Universal Robots PolyScope program: paganini.urp

Program paganini (installation=string_planes directory=/programs/hard_coded_pieces createdIn=5.17.3 lastSavedIn=5.17.3 robotSerialNumber=20245501435)
Calibrated DH parameters: a=[0.000154, -0.137004, -0.385524, -0.00002, 0.000092, 0]; d=[0.162441, 211.794786, -230.585024, 18.923638, 0.099786, 0.09951]; alpha=[1.569493, -0.001902, 0.003874, 1.570111, -1.570167, 0]; deltaTheta=[0, -1.242934, 1.056292, 0.186646, 0.000002, 0.000001]
InitVariablesNode
Robot Program (runOnlyOnce=true)
  SuppressedNode
    Wait Sleep waitTime=30
  Timer (action=Start) variable(name=beats)
  MoveL speed 600 mm/s, acceleration 1000 mm/s^2 (useActiveTCP=true) feature=Base
    Waypoint a_tip: TCP in base x=525.206 y=350.983 z=214.78 mm, rx=-1.3698 ry=-2.3362 rz=1.327 rad; joints [-161.028, -44.56, 81.191, -78.693, -115.03, -178.818] deg; TCP offset x=28.21 y=-96.107 z=-99.69 mm, rx=0 ry=0 rz=0 rad
    Waypoint a_frog: TCP in base x=336.638 y=773.336 z=103.937 mm, rx=-1.3698 ry=-2.3362 rz=1.327 rad; joints [-127.102, -6.181, 18.995, -50.118, -88.699, -156.884] deg
      Until EXPRESSION (allowActions=false) ExpressionBranch=beats≥1
    SuppressedNode
      Popup Message (haltProgram=false inputType=Variable) variable=beats
    Timer (action=Reset) variable=beats
  MoveL speed 150 mm/s, acceleration 400 mm/s^2 (useActiveTCP=true) feature=Base
    Waypoint a_tip: TCP in base x=525.206 y=350.983 z=214.78 mm, rx=-1.3698 ry=-2.3362 rz=1.327 rad; joints [-161.028, -44.56, 81.191, -78.693, -115.03, -178.818] deg
      Until EXPRESSION (allowActions=false) ExpressionBranch=beats≥2.5
    Timer (action=Reset) variable=beats
  MoveL speed 200 mm/s, acceleration 1200 mm/s^2 (useActiveTCP=true) feature=Base
    Waypoint a_tip: TCP in base x=525.206 y=350.983 z=214.78 mm, rx=-1.3698 ry=-2.3362 rz=1.327 rad; joints [-161.028, -44.56, 81.191, -78.693, -115.03, -178.818] deg
      Until EXPRESSION (allowActions=false) ExpressionBranch=beats≥0.75
    Timer (action=Reset) variable=beats
  MoveL speed 150 mm/s, acceleration 400 mm/s^2 (useActiveTCP=true) feature=Base
    Waypoint a_frog: TCP in base x=336.638 y=773.336 z=103.937 mm, rx=-1.3698 ry=-2.3362 rz=1.327 rad; joints [-127.102, -6.181, 18.995, -50.118, -88.699, -156.884] deg
      Until EXPRESSION (allowActions=false) ExpressionBranch=beats≥2.5
    Timer (action=Reset) variable=beats
  MoveL speed 250 mm/s, acceleration 1200 mm/s^2 (useActiveTCP=true) feature=Base
    Waypoint a_frog: TCP in base x=336.638 y=773.336 z=103.937 mm, rx=-1.3698 ry=-2.3362 rz=1.327 rad; joints [-127.102, -6.181, 18.995, -50.118, -88.699, -156.884] deg
      Until EXPRESSION (allowActions=false) ExpressionBranch=beats≥0.75
    Timer (action=Reset) variable=beats
  MoveL speed 250 mm/s, acceleration 1200 mm/s^2 (useActiveTCP=true) feature=Base
    Waypoint a_tip: TCP in base x=525.206 y=350.983 z=214.78 mm, rx=-1.3698 ry=-2.3362 rz=1.327 rad; joints [-161.028, -44.56, 81.191, -78.693, -115.03, -178.818] deg
      Until EXPRESSION (allowActions=false) ExpressionBranch=beats≥0.75
    Timer (action=Reset) variable=beats
  MoveJ speed 100 deg/s, acceleration 100 deg/s^2 (useActiveTCP=true) feature=Base
    Waypoint a_frog: TCP in base x=336.638 y=773.336 z=103.937 mm, rx=-1.3698 ry=-2.3362 rz=1.327 rad; joints [-127.102, -6.181, 18.995, -50.118, -88.699, -156.884] deg
  Timer (action=Reset) variable=beats
  MoveL speed 200 mm/s, acceleration 200 mm/s^2 (useActiveTCP=true) feature=Base
    Waypoint a_tip: TCP in base x=525.206 y=350.983 z=214.78 mm, rx=-1.3698 ry=-2.3362 rz=1.327 rad; joints [-161.028, -44.56, 81.191, -78.693, -115.03, -178.818] deg
      Until EXPRESSION (allowActions=false) ExpressionBranch=beats≥3
    Timer (action=Reset) variable=beats
  MoveL speed 600 mm/s, acceleration 1000 mm/s^2 (useActiveTCP=true) feature=Base
    Waypoint a_frog: TCP in base x=336.638 y=773.336 z=103.937 mm, rx=-1.3698 ry=-2.3362 rz=1.327 rad; joints [-127.102, -6.181, 18.995, -50.118, -88.699, -156.884] deg
      Until EXPRESSION (allowActions=false) ExpressionBranch=beats≥1
    Timer (action=Reset) variable=beats
  MoveL speed 150 mm/s, acceleration 400 mm/s^2 (useActiveTCP=true) feature=Base
    Waypoint a_tip: TCP in base x=525.206 y=350.983 z=214.78 mm, rx=-1.3698 ry=-2.3362 rz=1.327 rad; joints [-161.028, -44.56, 81.191, -78.693, -115.03, -178.818] deg
      Until EXPRESSION (allowActions=false) ExpressionBranch=beats≥2.5
    Timer (action=Reset) variable=beats
  MoveL speed 250 mm/s, acceleration 1200 mm/s^2 (useActiveTCP=true) feature=Base
    Waypoint a_tip: TCP in base x=525.206 y=350.983 z=214.78 mm, rx=-1.3698 ry=-2.3362 rz=1.327 rad; joints [-161.028, -44.56, 81.191, -78.693, -115.03, -178.818] deg
      Until EXPRESSION (allowActions=false) ExpressionBranch=beats≥0.75
    Timer (action=Reset) variable=beats
  MoveL speed 150 mm/s, acceleration 400 mm/s^2 (useActiveTCP=true) feature=Base
    Waypoint a_frog: TCP in base x=336.638 y=773.336 z=103.937 mm, rx=-1.3698 ry=-2.3362 rz=1.327 rad; joints [-127.102, -6.181, 18.995, -50.118, -88.699, -156.884] deg
      Until EXPRESSION (allowActions=false) ExpressionBranch=beats≥1.5
    Timer (action=Reset) variable=beats
  MoveL speed 250 mm/s, acceleration 1200 mm/s^2 (useActiveTCP=true) feature=Base
    Waypoint a_tip: TCP in base x=525.206 y=350.983 z=214.78 mm, rx=-1.3698 ry=-2.3362 rz=1.327 rad; joints [-161.028, -44.56, 81.191, -78.693, -115.03, -178.818] deg
      Until EXPRESSION (allowActions=false) ExpressionBranch=beats≥0.75
    Timer (action=Reset) variable=beats
  MoveL speed 150 mm/s, acceleration 400 mm/s^2 (useActiveTCP=true) feature=Base
    Waypoint a_frog: TCP in base x=336.638 y=773.336 z=103.937 mm, rx=-1.3698 ry=-2.3362 rz=1.327 rad; joints [-127.102, -6.181, 18.995, -50.118, -88.699, -156.884] deg
      Until EXPRESSION (allowActions=false) ExpressionBranch=beats≥1.5
    Timer (action=Reset) variable=beats
  MoveL speed 250 mm/s, acceleration 1200 mm/s^2 (useActiveTCP=true) feature=Base
    Waypoint a_frog: TCP in base x=336.638 y=773.336 z=103.937 mm, rx=-1.3698 ry=-2.3362 rz=1.327 rad; joints [-127.102, -6.181, 18.995, -50.118, -88.699, -156.884] deg
      Until EXPRESSION (allowActions=false) ExpressionBranch=beats≥0.75
    Timer (action=Reset) variable=beats
  MoveL speed 100 mm/s, acceleration 150 mm/s^2 (useActiveTCP=true) feature=Base
    Waypoint a_tip: TCP in base x=525.206 y=350.983 z=214.78 mm, rx=-1.3698 ry=-2.3362 rz=1.327 rad; joints [-161.028, -44.56, 81.191, -78.693, -115.03, -178.818] deg
      Until EXPRESSION (allowActions=false) ExpressionBranch=beats≥3
    Timer (action=Reset) variable=beats
  MoveL speed 150 mm/s, acceleration 200 mm/s^2 (useActiveTCP=true) feature=Base
    Waypoint a_tip: TCP in base x=525.206 y=350.983 z=214.78 mm, rx=-1.3698 ry=-2.3362 rz=1.327 rad; joints [-161.028, -44.56, 81.191, -78.693, -115.03, -178.818] deg
      Until EXPRESSION (allowActions=false) ExpressionBranch=beats≥1
    Timer (action=Reset) variable=beats
  MoveL speed 700 mm/s, acceleration 1200 mm/s^2 (useActiveTCP=true) feature=Base
    Waypoint a_frog: TCP in base x=336.638 y=773.336 z=103.937 mm, rx=-1.3698 ry=-2.3362 rz=1.327 rad; joints [-127.102, -6.181, 18.995, -50.118, -88.699, -156.884] deg
      Until EXPRESSION (allowActions=false) ExpressionBranch=beats≥1
    Timer (action=Reset) variable=beats
  SuppressedNode
    Wait Sleep waitTime=30
  MoveL speed 150 mm/s, acceleration 400 mm/s^2 (useActiveTCP=true) feature=Base
    Waypoint a_tip: TCP in base x=525.206 y=350.983 z=214.78 mm, rx=-1.3698 ry=-2.3362 rz=1.327 rad; joints [-161.028, -44.56, 81.191, -78.693, -115.03, -178.818] deg
      Until EXPRESSION (allowActions=false) ExpressionBranch=beats≥2.5
    Timer (action=Reset) variable=beats
  MoveL speed 200 mm/s, acceleration 1200 mm/s^2 (useActiveTCP=true) feature=Base
    Waypoint a_tip: TCP in base x=525.206 y=350.983 z=214.78 mm, rx=-1.3698 ry=-2.3362 rz=1.327 rad; joints [-161.028, -44.56, 81.191, -78.693, -115.03, -178.818] deg
      Until EXPRESSION (allowActions=false) ExpressionBranch=beats≥0.75
    Timer (action=Reset) variable=beats
  MoveL speed 150 mm/s, acceleration 400 mm/s^2 (useActiveTCP=true) feature=Base
    Waypoint a_frog: TCP in base x=336.638 y=773.336 z=103.937 mm, rx=-1.3698 ry=-2.3362 rz=1.327 rad; joints [-127.102, -6.181, 18.995, -50.118, -88.699, -156.884] deg
      Until EXPRESSION (allowActions=false) ExpressionBranch=beats≥2.5
    Timer (action=Reset) variable=beats
  MoveL speed 250 mm/s, acceleration 1200 mm/s^2 (useActiveTCP=true) feature=Base
    Waypoint a_frog: TCP in base x=336.638 y=773.336 z=103.937 mm, rx=-1.3698 ry=-2.3362 rz=1.327 rad; joints [-127.102, -6.181, 18.995, -50.118, -88.699, -156.884] deg
      Until EXPRESSION (allowActions=false) ExpressionBranch=beats≥0.75
    Timer (action=Reset) variable=beats
  MoveL speed 250 mm/s, acceleration 1200 mm/s^2 (useActiveTCP=true) feature=Base
    Waypoint a_tip: TCP in base x=525.206 y=350.983 z=214.78 mm, rx=-1.3698 ry=-2.3362 rz=1.327 rad; joints [-161.028, -44.56, 81.191, -78.693, -115.03, -178.818] deg
      Until EXPRESSION (allowActions=false) ExpressionBranch=beats≥0.75
    Timer (action=Reset) variable=beats
  MoveJ speed 100 deg/s, acceleration 100 deg/s^2 (useActiveTCP=true) feature=Base
    Waypoint a_frog: TCP in base x=336.638 y=773.336 z=103.937 mm, rx=-1.3698 ry=-2.3362 rz=1.327 rad; joints [-127.102, -6.181, 18.995, -50.118, -88.699, -156.884] deg
  Timer (action=Reset) variable=beats
  MoveL speed 200 mm/s, acceleration 200 mm/s^2 (useActiveTCP=true) feature=Base
    Waypoint a_tip: TCP in base x=525.206 y=350.983 z=214.78 mm, rx=-1.3698 ry=-2.3362 rz=1.327 rad; joints [-161.028, -44.56, 81.191, -78.693, -115.03, -178.818] deg
      Until EXPRESSION (allowActions=false) ExpressionBranch=beats≥3
    Timer (action=Reset) variable=beats
  MoveL speed 600 mm/s, acceleration 1000 mm/s^2 (useActiveTCP=true) feature=Base
    Waypoint a_frog: TCP in base x=336.638 y=773.336 z=103.937 mm, rx=-1.3698 ry=-2.3362 rz=1.327 rad; joints [-127.102, -6.181, 18.995, -50.118, -88.699, -156.884] deg
      Until EXPRESSION (allowActions=false) ExpressionBranch=beats≥1
    Timer (action=Reset) variable=beats
  MoveL speed 150 mm/s, acceleration 400 mm/s^2 (useActiveTCP=true) feature=Base
    Waypoint a_tip: TCP in base x=525.206 y=350.983 z=214.78 mm, rx=-1.3698 ry=-2.3362 rz=1.327 rad; joints [-161.028, -44.56, 81.191, -78.693, -115.03, -178.818] deg
      Until EXPRESSION (allowActions=false) ExpressionBranch=beats≥2.5
    Timer (action=Reset) variable=beats
  MoveL speed 250 mm/s, acceleration 1200 mm/s^2 (useActiveTCP=true) feature=Base
    Waypoint a_frog: TCP in base x=336.638 y=773.336 z=103.937 mm, rx=-1.3698 ry=-2.3362 rz=1.327 rad; joints [-127.102, -6.181, 18.995, -50.118, -88.699, -156.884] deg
      Until EXPRESSION (allowActions=false) ExpressionBranch=beats≥0.75
    Timer (action=Reset) variable=beats
  MoveL speed 150 mm/s, acceleration 400 mm/s^2 (useActiveTCP=true) feature=Base
    Waypoint a_tip: TCP in base x=525.206 y=350.983 z=214.78 mm, rx=-1.3698 ry=-2.3362 rz=1.327 rad; joints [-161.028, -44.56, 81.191, -78.693, -115.03, -178.818] deg
      Until EXPRESSION (allowActions=false) ExpressionBranch=beats≥1.5
    Timer (action=Reset) variable=beats
  MoveL speed 250 mm/s, acceleration 1200 mm/s^2 (useActiveTCP=true) feature=Base
    Waypoint a_frog: TCP in base x=336.638 y=773.336 z=103.937 mm, rx=-1.3698 ry=-2.3362 rz=1.327 rad; joints [-127.102, -6.181, 18.995, -50.118, -88.699, -156.884] deg
      Until EXPRESSION (allowActions=false) ExpressionBranch=beats≥0.75
    Timer (action=Reset) variable=beats
  MoveL speed 400 mm/s, acceleration 800 mm/s^2 (useActiveTCP=true) feature=Base
    Waypoint a_tip: TCP in base x=525.206 y=350.983 z=214.78 mm, rx=-1.3698 ry=-2.3362 rz=1.327 rad; joints [-161.028, -44.56, 81.191, -78.693, -115.03, -178.818] deg
      Until EXPRESSION (allowActions=false) ExpressionBranch=beats≥2
    Timer (action=Reset) variable=beats
  MoveL speed 150 mm/s, acceleration 200 mm/s^2 (useActiveTCP=true) feature=Base
    Waypoint a_frog: TCP in base x=336.638 y=773.336 z=103.937 mm, rx=-1.3698 ry=-2.3362 rz=1.327 rad; joints [-127.102, -6.181, 18.995, -50.118, -88.699, -156.884] deg
      Until EXPRESSION (allowActions=false) ExpressionBranch=beats≥3
    Timer (action=Reset) variable=beats
